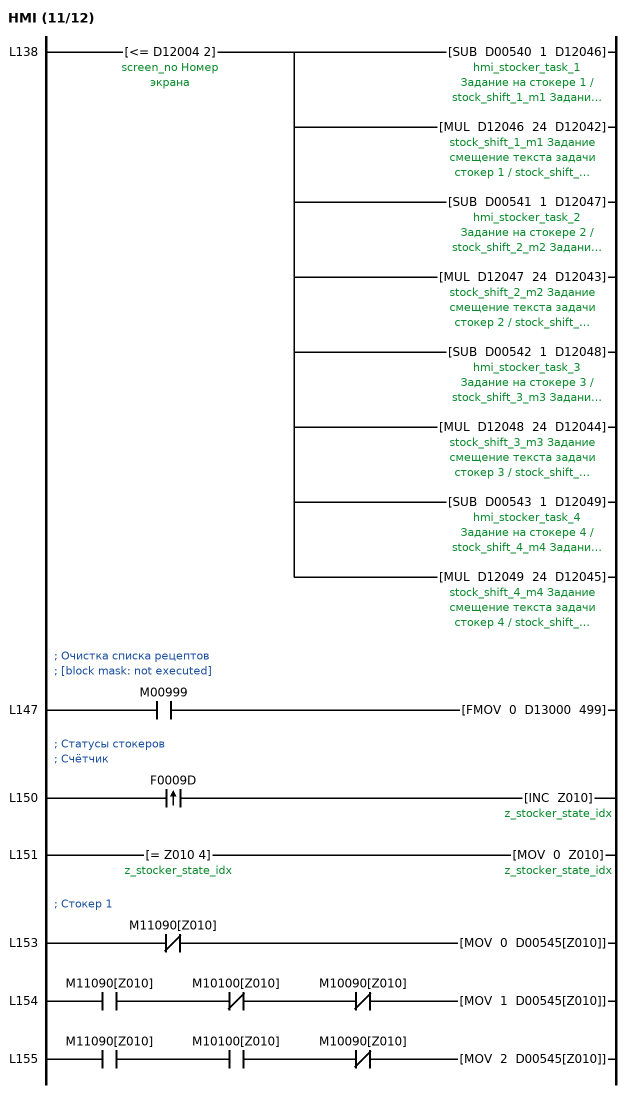
; L138
LOAD<=    D12004 2	// screen_no Номер экрана
SUB       D00540 1 D12046	// hmi_stocker_task_1 Задание на стокере 1 / stock_shift_1_m1 Задание смещение текста задачи стокер 1
MUL       D12046 24 D12042	// stock_shift_1_m1 Задание смещение текста задачи стокер 1 / stock_shift_1 Задание смещение текста задачи стокер 1
SUB       D00541 1 D12047	// hmi_stocker_task_2 Задание на стокере 2 / stock_shift_2_m2 Задание смещение текста задачи стокер 2
MUL       D12047 24 D12043	// stock_shift_2_m2 Задание смещение текста задачи стокер 2 / stock_shift_2 Задание смещение текста задачи стокер 2
SUB       D00542 1 D12048	// hmi_stocker_task_3 Задание на стокере 3 / stock_shift_3_m3 Задание смещение текста задачи стокер 3
MUL       D12048 24 D12044	// stock_shift_3_m3 Задание смещение текста задачи стокер 3 / stock_shift_3 Задание смещение текста задачи стокер 3
SUB       D00543 1 D12049	// hmi_stocker_task_4 Задание на стокере 4 / stock_shift_4_m4 Задание смещение текста задачи стокер 4
MUL       D12049 24 D12045	// stock_shift_4_m4 Задание смещение текста задачи стокер 4 / stock_shift_4 Задание смещение текста задачи стокер 4
// Очистка списка рецептов
; L147 (block mask: not executed)
LOAD      M00999
FMOV      0 D13000 499
// Статусы стокеров
// Счётчик
; L150
LOADP     F0009D
INC       Z010	// z_stocker_state_idx
; L151
LOAD=     Z010 4	// z_stocker_state_idx
MOV       0 Z010	// z_stocker_state_idx
// Стокер 1
; L153
LOAD NOT  M11090[Z010]
MOV       0 D00545[Z010]
; L154
LOAD      M11090[Z010]
AND NOT   M10100[Z010]
AND NOT   M10090[Z010]
MOV       1 D00545[Z010]
; L155
LOAD      M11090[Z010]
AND       M10100[Z010]
AND NOT   M10090[Z010]
MOV       2 D00545[Z010]

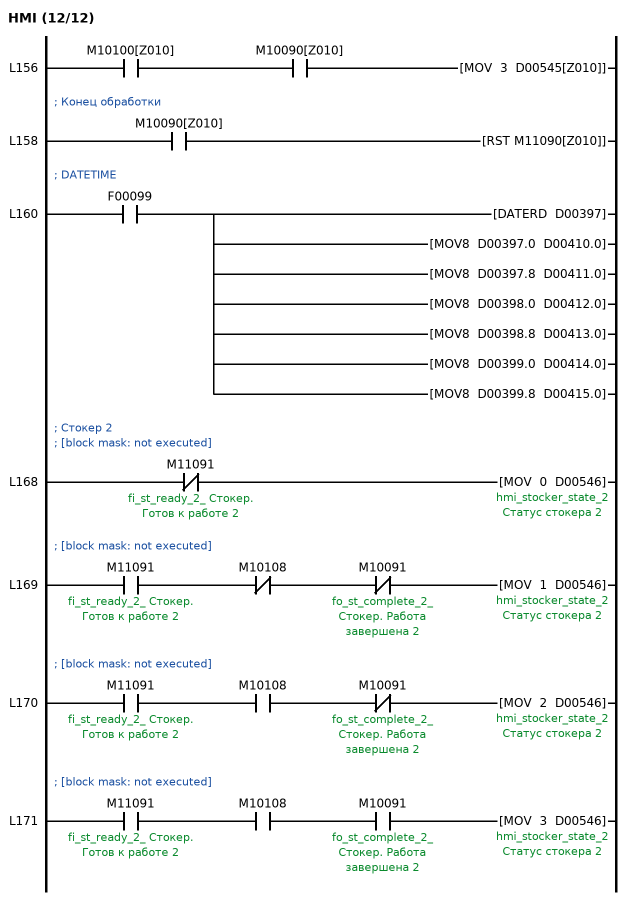
; L156
LOAD      M10100[Z010]
AND       M10090[Z010]
MOV       3 D00545[Z010]
// Конец обработки
; L158
LOAD      M10090[Z010]
RST       M11090[Z010]
// DATETIME
; L160
LOAD      F00099
DATERD    D00397
MOV8      D00397.0 D00410.0
MOV8      D00397.8 D00411.0
MOV8      D00398.0 D00412.0
MOV8      D00398.8 D00413.0
MOV8      D00399.0 D00414.0
MOV8      D00399.8 D00415.0
// Стокер 2
; L168 (block mask: not executed)
LOAD NOT  M11091	// fi_st_ready_2_ Стокер. Готов к работе 2
MOV       0 D00546	// hmi_stocker_state_2 Статус стокера 2
; L169 (block mask: not executed)
LOAD      M11091	// fi_st_ready_2_ Стокер. Готов к работе 2
AND NOT   M10108
AND NOT   M10091	// fo_st_complete_2_ Стокер. Работа завершена 2
MOV       1 D00546	// hmi_stocker_state_2 Статус стокера 2
; L170 (block mask: not executed)
LOAD      M11091	// fi_st_ready_2_ Стокер. Готов к работе 2
AND       M10108
AND NOT   M10091	// fo_st_complete_2_ Стокер. Работа завершена 2
MOV       2 D00546	// hmi_stocker_state_2 Статус стокера 2
; L171 (block mask: not executed)
LOAD      M11091	// fi_st_ready_2_ Стокер. Готов к работе 2
AND       M10108
AND       M10091	// fo_st_complete_2_ Стокер. Работа завершена 2
MOV       3 D00546	// hmi_stocker_state_2 Статус стокера 2

PROGRAM ERROR (task: Scan Program)

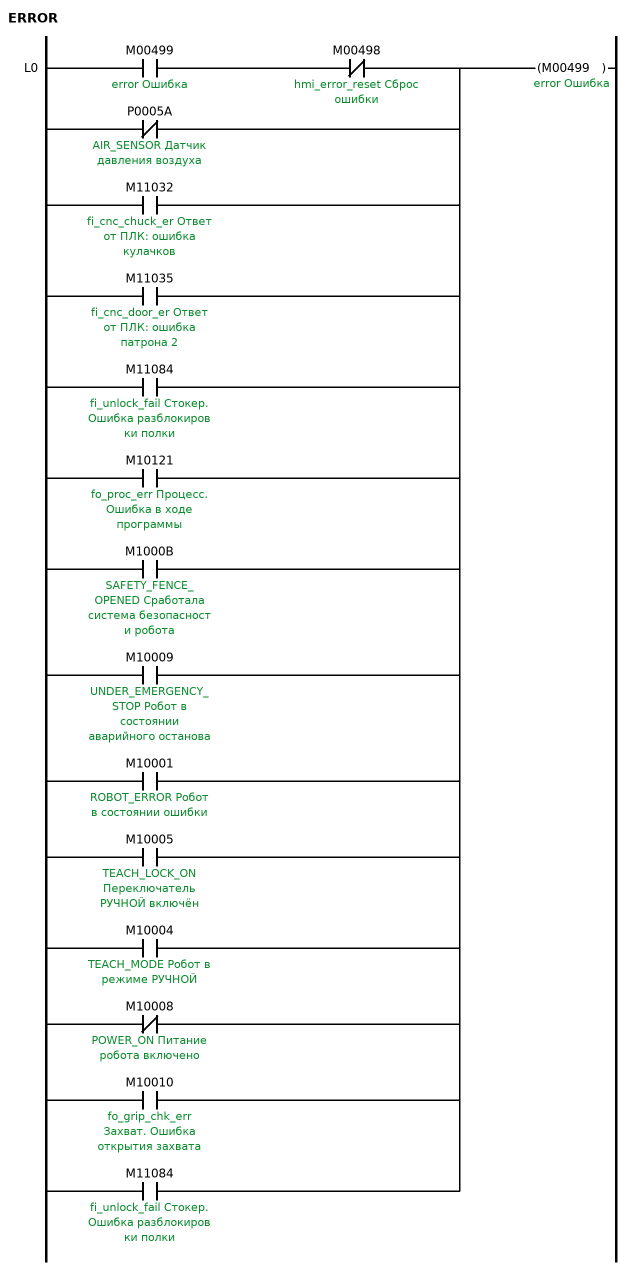
; L0
LOAD      M00499	// error Ошибка
AND NOT   M00498	// hmi_error_reset Сброс ошибки
OR NOT    P0005A	// AIR_SENSOR Датчик давления воздуха
OR        M11032	// fi_cnc_chuck_er Ответ от ПЛК: ошибка кулачков
OR        M11035	// fi_cnc_door_er Ответ от ПЛК: ошибка патрона 2
OR        M11084	// fi_unlock_fail Стокер. Ошибка разблокировки полки
OR        M10121	// fo_proc_err Процесс. Ошибка в ходе программы
OR        M1000B	// SAFETY_FENCE_OPENED Сработала система безопасности робота
OR        M10009	// UNDER_EMERGENCY_STOP Робот в состоянии аварийного останова
OR        M10001	// ROBOT_ERROR Робот в состоянии ошибки
OR        M10005	// TEACH_LOCK_ON Переключатель РУЧНОЙ включён
OR        M10004	// TEACH_MODE Робот в режиме РУЧНОЙ
OR NOT    M10008	// POWER_ON Питание робота включено
OR        M10010	// fo_grip_chk_err Захват. Ошибка открытия захвата
OR        M11084	// fi_unlock_fail Стокер. Ошибка разблокировки полки
OUT       M00499	// error Ошибка

VARIABLES AND COMMENTS (devices not used above)
M1000C	BIT	BATTERY_ALARM // Батарейка энкодеров садится
M00546	BIT	CMD_CHUCK_CLOSE // Закрыть патрон 1
P00092	BIT	CMD_LAST // Последняя деталь
P00091	BIT	CMD_RBTALM // Ошибка робота
M00513	BIT	cnc_chuck_close_flag // Флаг закрытия кулачков
M00512	BIT	cnc_chuck_open_flag // Флаг открытия кулачков
P00044	BIT	CNC_DOOR_CLOSED // Патрон 2 закрыт
P00043	BIT	CNC_DOOR_OPENED // Патрон 2 открыт
P0005F	BIT	CNC_PG_NG // Ошибка поиска программы
P00046	BIT	CNC_PG_OK // Поиск программы успешен
D00200	WORD	current_stocker
P0008F	BIT	EMPTY
M11001	BIT	EXT_ERROR_RESET // Сбросить ошибку на роботе
M11037	BIT	fi_cnc_blocked // Ответ от ПЛК: станок заблокирован
M11034	BIT	fi_cnc_door_cl // Ответ от ПЛК: патрон 2 закрыта
M11033	BIT	fi_cnc_door_op // Ответ от ПЛК: патрон 2 открыт
M1107F	BIT	fi_cnc_pick_ovp_7_ // Станок. Прижим при взятии бит 7
M11077	BIT	fi_cnc_put_ovp_7_ // Станок. Прижим при установке бит 7
M11150	BIT	fi_de_data_0_ // Обмен данными. Данные бит 0
M1115F	BIT	fi_de_data_15_ // Обмен данными. Данные бит 15
M11137	BIT	fi_de_recipe_7_ // Обмен данными. Тип рецепта бит 7
M11147	BIT	fi_de_table_el_7_ // Обмен данными. Элемент таблицы бит 7
M1113F	BIT	fi_de_table_id_7_ // Обмен данными. Номер таблицы бит 7
M11010	BIT	fi_grip_check // Захват. Проверять ли датчик открытия захвата
M11012	BIT	fi_grip_close_1_ // Захват. Закрыть захват 1
M11014	BIT	fi_grip_close_2_ // Захват. Закрыть захват 2
M1102F	BIT	fi_grip_ctime_7_ // Захват. Время на закрытие захвата бит 7
M1101C	BIT	fi_grip_etime_7_ // Захват. Время проверки захвата бит 7
M11011	BIT	fi_grip_open_1_ // Захват. Открыть захват 1
M11013	BIT	fi_grip_open_2_ // Захват. Открыть захват 2
M11027	BIT	fi_grip_otime_7_ // Захват. Время на открытие захвата бит 7
M11160	BIT	fi_mon_speed_0_ // Робот. Множитель скорости  бит 0
M11167	BIT	fi_mon_speed_7_ // Робот. Множитель скорости  бит 7
M11120	BIT	fi_proc_start // Процесс. Запуск процесса / продолжить процесс
M11127	BIT	fi_robot_pgreset // Сброс цикла
M11090	BIT	fi_st_ready_1_ // Стокер. Готов к работе 1
M11092	BIT	fi_st_ready_3_ // Стокер. Готов к работе 3
M11093	BIT	fi_st_ready_4_ // Стокер. Готов к работе 4
M1108F	BIT	fi_st_search // Стокер. Активировать подсчёт заготовок
M11107	BIT	fi_st_task_1__7_ // Процесс. Задание на стокере 1 бит 7
M1110F	BIT	fi_st_task_2__7_ // Процесс. Задание на стокере 2 бит 7
M11117	BIT	fi_st_task_3__7_ // Процесс. Задание на стокере 3 бит 7
M1111F	BIT	fi_st_task_4__7_ // Процесс. Задание на стокере 4 бит 7
M11040	BIT	fi_x_cor_cnc_0_ // Станок. Корректировка патрона по оси Х бит 0
M1104F	BIT	fi_x_cor_cnc_15_ // Станок. Корректировка патрона по оси Х бит 15
M11050	BIT	fi_y_cor_cnc_0_ // Станок. Корректировка патрона по оси Y бит 0
M1105F	BIT	fi_y_cor_cnc_15_ // Станок. Корректировка патрона по оси Y бит 15
M11060	BIT	fi_z_cor_cnc_0_ // Станок. Корректировка патрона по оси Z бит 0
M1106F	BIT	fi_z_cor_cnc_15_ // Станок. Корректировка патрона по оси Z бит 15
M12022	BIT	flag_load_type_6 // Флаг загруить элемент типа 6
M12023	BIT	flag_load_type_7 // Флаг загруить элемент типа 7
M12024	BIT	flag_load_type_8 // Флаг загруить элемент типа 8
M1201A	BIT	flag_save_type_6 // Флаг сохранить элемент типа 6
M1201B	BIT	flag_save_type_7 // Флаг сохранить элемент типа 7
M1201C	BIT	flag_save_type_8 // Флаг сохранить элемент типа 8
M10037	BIT	fo_cnc_block // Команда станку - заблокировать
M1003F	BIT	fo_cnc_pg_7_ // Команда станку - бит программы 7
M10012	BIT	fo_grip_closed_1_ // Захват. Захват 1 закрыт
M10014	BIT	fo_grip_closed_2_ // Захват. Захват 2 закрыт
M10011	BIT	fo_grip_opened_1_ // Захват. Захват 1 открыт
M10013	BIT	fo_grip_opened_2_ // Захват. Захват 2 открыт
M10015	BIT	fo_grip_sensor // Захват. Датчик заготовки
M10120	BIT	fo_proc_on // Процесс. Процесс запущен
M10090	BIT	fo_st_complete_1_ // Стокер. Работа завершена 1
M10092	BIT	fo_st_complete_3_ // Стокер. Работа завершена 3
M10093	BIT	fo_st_complete_4_ // Стокер. Работа завершена 4
M10085	BIT	fo_st_opened_1_ // Стокер. Открыт 1
M10086	BIT	fo_st_opened_2_ // Стокер. Открыт 2
M10087	BIT	fo_st_opened_3_ // Стокер. Открыт 3
M10088	BIT	fo_st_opened_4_ // Стокер. Открыт 4
M00551	BIT	hmi_air_off
D00512	WORD	hmi_chuck_close_time // Время на закрытие кулачков
D00513	WORD	hmi_chuck_err_time // Время ошибки кулачков
D00511	WORD	hmi_chuck_open_time // Время на открытие кулачков
M0050A	BIT	hmi_cnc_chuck_close_check // Проверять датчик закрытия кулачков станка
M00509	BIT	hmi_cnc_chuck_open_check // Проверять датчик открытия кулачков станка
M0050E	BIT	hmi_cnc_door_close_check // Проверять датчик закрытия патрона 2 станка
M0050D	BIT	hmi_cnc_door_open_check // Проверять датчик открытия патрона 2 станка
M00516	BIT	hmi_cnc_lock // Команда станку с HMI  - заблокировать
D00522	WORD	hmi_cnc_pick_ovlp // Оверлап при взятии 
D00523	WORD	hmi_cnc_put_ovlp // Оверлап при заборе
M00517	BIT	hmi_cnc_unlock // Команда станку с HMI  - разблокировать
D00519	WORD	hmi_cnc_x_cor // Корректировка точки станка Х
D00520	WORD	hmi_cnc_y_cor // Корректировка точки станка Y
D00521	WORD	hmi_cnc_z_cor // Корректировка точки станка Z
M0052B	BIT	hmi_door_chuck_close // Лампа Датчик закрытия патрона 2
M0052A	BIT	hmi_door_chuck_open // Лампа Датчик открытия патрона 2
D00516	WORD	hmi_door_close_time // Время на закрытие патрона 2
D00517	WORD	hmi_door_err_time // Время ошибки патрона 2
D00515	WORD	hmi_door_open_time // Время на открытие патрона 2
M00529	BIT	hmi_lamp_chuck_close // Лампа Датчик закрытия кулачков
M00528	BIT	hmi_lamp_chuck_open // Лампа Датчик открытия кулачков
M00525	BIT	hmi_robot_process_on // Запуск процесса обработки 
M00526	BIT	hmi_robot_process_stop // Остановка процесса обработки 
M00506	BIT	hmi_robot_slow // Замедление робота при приближении
D12624.0	BIT	hmi_shaft_back // Требуется ли возврат вала в кондуктор
D00534	WORD	hmi_stocker_open_delay // Задержка при открытии стокера
D00545	WORD	hmi_stocker_state_1 // Статус стокера 1
D00547	WORD	hmi_stocker_state_3 // Статус стокера 3
D00548	WORD	hmi_stocker_state_4 // Статус стокера 4
M10006	BIT	HOME // Робот в домашнем положении 1
M10007	BIT	HOME2 // Робот в домашнем положении 2
D12050	WORD	plate_name_shift // Смещение имени пластины коррекция
D12051	WORD	plate_name_shift_m1 // Смещение имени пластины коррекция
D00500	WORD	plc_power_errors // Количество включений ПЛК 
D12001	WORD	recipe_error_code // Код ошибки рецепта
M12002	BIT	recipe_state_ok // Рецепт сохранён/загружен
M12012	BIT	save_ok_type_6 // Элемент сохранён тип 6
M12013	BIT	save_ok_type_7 // Элемент сохранён тип 7
M12014	BIT	save_ok_type_8 // Элемент сохранён тип 8
M1200A	BIT	save_type_6 // Сохранить элемент типа 6
M1200B	BIT	save_type_7 // Сохранить элемент типа 7
M1200C	BIT	save_type_8 // Сохранить элемент типа 8
M00000	BIT	start_task
T0560	BIT/WORD	T100_data_ready_1 // Таймер на подготовку данных 1
T0561	BIT/WORD	T100_data_ready_2 // Таймер на подготовку данных 2
T0562	BIT/WORD	T100_data_ready_3 // Таймер на подготовку данных 3
T0563	BIT/WORD	T100_data_ready_4 // Таймер на подготовку данных 4
T0564	BIT/WORD	T100_data_ready_5 // Таймер на подготовку данных 5
T0565	BIT/WORD	T100_data_ready_6 // Таймер на подготовку данных 6
T0566	BIT/WORD	T100_data_ready_7 // Таймер на подготовку данных 7
T0921	BIT/WORD	T100_load_delay_6 // Таймаут на загрузку 6
T0922	BIT/WORD	T100_load_delay_7 // Таймаут на загрузку 7
T0913	BIT/WORD	T100_save_delay_6 // Время сохранения 6
T0914	BIT/WORD	T100_save_delay_7 // Время сохранения 7
T0915	BIT/WORD	T100_save_delay_8 // Время сохранения 8
M00001	BIT	work_stocker_1
M00002	BIT	work_stocker_2
M00003	BIT	work_stocker_3
M00004	BIT	work_stocker_4
M10039	BIT	Команда станку - бит программы 1
M1003A	BIT	Команда станку - бит программы 2
M1003B	BIT	Команда станку - бит программы 3
M1003C	BIT	Команда станку - бит программы 4
M1003D	BIT	Команда станку - бит программы 5
M1003E	BIT	Команда станку - бит программы 6
M11016	BIT	Захват. Время проверки захвата бит 1
M11017	BIT	Захват. Время проверки захвата бит 2
M11018	BIT	Захват. Время проверки захвата бит 3
M11019	BIT	Захват. Время проверки захвата бит 4
M1101A	BIT	Захват. Время проверки захвата бит 5
M1101B	BIT	Захват. Время проверки захвата бит 6
M11021	BIT	Захват. Время на открытие захвата бит 1
M11022	BIT	Захват. Время на открытие захвата бит 2
M11023	BIT	Захват. Время на открытие захвата бит 3
M11024	BIT	Захват. Время на открытие захвата бит 4
M11025	BIT	Захват. Время на открытие захвата бит 5
M11026	BIT	Захват. Время на открытие захвата бит 6
M11029	BIT	Захват. Время на закрытие захвата бит 1
M1102A	BIT	Захват. Время на закрытие захвата бит 2
M1102B	BIT	Захват. Время на закрытие захвата бит 3
M1102C	BIT	Захват. Время на закрытие захвата бит 4
M1102D	BIT	Захват. Время на закрытие захвата бит 5
M1102E	BIT	Захват. Время на закрытие захвата бит 6
M11041	BIT	Станок. Корректировка патрона по оси Х бит 1
M11042	BIT	Станок. Корректировка патрона по оси Х бит 2
M11043	BIT	Станок. Корректировка патрона по оси Х бит 3
M11044	BIT	Станок. Корректировка патрона по оси Х бит 4
M11045	BIT	Станок. Корректировка патрона по оси Х бит 5
M11046	BIT	Станок. Корректировка патрона по оси Х бит 6
M11047	BIT	Станок. Корректировка патрона по оси Х бит 7
M11048	BIT	Станок. Корректировка патрона по оси Х бит 8
M11049	BIT	Станок. Корректировка патрона по оси Х бит 9
M1104A	BIT	Станок. Корректировка патрона по оси Х бит 10
M1104B	BIT	Станок. Корректировка патрона по оси Х бит 11
M1104C	BIT	Станок. Корректировка патрона по оси Х бит 12
M1104D	BIT	Станок. Корректировка патрона по оси Х бит 13
M1104E	BIT	Станок. Корректировка патрона по оси Х бит 14
M11051	BIT	Станок. Корректировка патрона по оси Y бит 1
M11052	BIT	Станок. Корректировка патрона по оси Y бит 2
M11053	BIT	Станок. Корректировка патрона по оси Y бит 3
M11054	BIT	Станок. Корректировка патрона по оси Y бит 4
M11055	BIT	Станок. Корректировка патрона по оси Y бит 5
M11056	BIT	Станок. Корректировка патрона по оси Y бит 6
M11057	BIT	Станок. Корректировка патрона по оси Y бит 7
M11058	BIT	Станок. Корректировка патрона по оси Y бит 8
M11059	BIT	Станок. Корректировка патрона по оси Y бит 9
M1105A	BIT	Станок. Корректировка патрона по оси Y бит 10
M1105B	BIT	Станок. Корректировка патрона по оси Y бит 11
M1105C	BIT	Станок. Корректировка патрона по оси Y бит 12
M1105D	BIT	Станок. Корректировка патрона по оси Y бит 13
M1105E	BIT	Станок. Корректировка патрона по оси Y бит 14
M11061	BIT	Станок. Корректировка патрона по оси Z бит 1
M11062	BIT	Станок. Корректировка патрона по оси Z бит 2
M11063	BIT	Станок. Корректировка патрона по оси Z бит 3
M11064	BIT	Станок. Корректировка патрона по оси Z бит 4
M11065	BIT	Станок. Корректировка патрона по оси Z бит 5
M11066	BIT	Станок. Корректировка патрона по оси Z бит 6
M11067	BIT	Станок. Корректировка патрона по оси Z бит 7
M11068	BIT	Станок. Корректировка патрона по оси Z бит 8
M11069	BIT	Станок. Корректировка патрона по оси Z бит 9
M1106A	BIT	Станок. Корректировка патрона по оси Z бит 10
M1106B	BIT	Станок. Корректировка патрона по оси Z бит 11
M1106C	BIT	Станок. Корректировка патрона по оси Z бит 12
M1106D	BIT	Станок. Корректировка патрона по оси Z бит 13
M1106E	BIT	Станок. Корректировка патрона по оси Z бит 14
M11071	BIT	Станок. Прижим при установке бит 1
M11072	BIT	Станок. Прижим при установке бит 2
M11073	BIT	Станок. Прижим при установке бит 3
M11074	BIT	Станок. Прижим при установке бит 4
M11075	BIT	Станок. Прижим при установке бит 5
M11076	BIT	Станок. Прижим при установке бит 6
M11079	BIT	Станок. Прижим при взятии бит 1
M1107A	BIT	Станок. Прижим при взятии бит 2
M1107B	BIT	Станок. Прижим при взятии бит 3
M1107C	BIT	Станок. Прижим при взятии бит 4
M1107D	BIT	Станок. Прижим при взятии бит 5
M1107E	BIT	Станок. Прижим при взятии бит 6
M11101	BIT	Процесс. Задание на стокере 1 бит 1
M11102	BIT	Процесс. Задание на стокере 1 бит 2
M11103	BIT	Процесс. Задание на стокере 1 бит 3
M11104	BIT	Процесс. Задание на стокере 1 бит 4
M11105	BIT	Процесс. Задание на стокере 1 бит 5
M11106	BIT	Процесс. Задание на стокере 1 бит 6
M11109	BIT	Процесс. Задание на стокере 2 бит 1
M1110A	BIT	Процесс. Задание на стокере 2 бит 2
M1110B	BIT	Процесс. Задание на стокере 2 бит 3
M1110C	BIT	Процесс. Задание на стокере 2 бит 4
M1110D	BIT	Процесс. Задание на стокере 2 бит 5
M1110E	BIT	Процесс. Задание на стокере 2 бит 6
M11111	BIT	Процесс. Задание на стокере 3 бит 1
M11112	BIT	Процесс. Задание на стокере 3 бит 2
M11113	BIT	Процесс. Задание на стокере 3 бит 3
M11114	BIT	Процесс. Задание на стокере 3 бит 4
M11115	BIT	Процесс. Задание на стокере 3 бит 5
M11116	BIT	Процесс. Задание на стокере 3 бит 6
M11119	BIT	Процесс. Задание на стокере 4 бит 1
M1111A	BIT	Процесс. Задание на стокере 4 бит 2
M1111B	BIT	Процесс. Задание на стокере 4 бит 3
M1111C	BIT	Процесс. Задание на стокере 4 бит 4
M1111D	BIT	Процесс. Задание на стокере 4 бит 5
M1111E	BIT	Процесс. Задание на стокере 4 бит 6
M11131	BIT	Обмен данными. Тип рецепта бит 1
M11132	BIT	Обмен данными. Тип рецепта бит 2
M11133	BIT	Обмен данными. Тип рецепта бит 3
M11134	BIT	Обмен данными. Тип рецепта бит 4
M11135	BIT	Обмен данными. Тип рецепта бит 5
M11136	BIT	Обмен данными. Тип рецепта бит 6
M11139	BIT	Обмен данными. Номер таблицы бит 1
M1113A	BIT	Обмен данными. Номер таблицы бит 2
M1113B	BIT	Обмен данными. Номер таблицы бит 3
M1113C	BIT	Обмен данными. Номер таблицы бит 4
M1113D	BIT	Обмен данными. Номер таблицы бит 5
M1113E	BIT	Обмен данными. Номер таблицы бит 6
M11141	BIT	Обмен данными. Элемент таблицы бит 1
M11142	BIT	Обмен данными. Элемент таблицы бит 2
M11143	BIT	Обмен данными. Элемент таблицы бит 3
M11144	BIT	Обмен данными. Элемент таблицы бит 4
M11145	BIT	Обмен данными. Элемент таблицы бит 5
M11146	BIT	Обмен данными. Элемент таблицы бит 6
M11151	BIT	Обмен данными. Данные бит 1
M11152	BIT	Обмен данными. Данные бит 2
M11153	BIT	Обмен данными. Данные бит 3
M11154	BIT	Обмен данными. Данные бит 4
M11155	BIT	Обмен данными. Данные бит 5
M11156	BIT	Обмен данными. Данные бит 6
M11157	BIT	Обмен данными. Данные бит 7
M11158	BIT	Обмен данными. Данные бит 8
M11159	BIT	Обмен данными. Данные бит 9
M1115A	BIT	Обмен данными. Данные бит 10
M1115B	BIT	Обмен данными. Данные бит 11
M1115C	BIT	Обмен данными. Данные бит 12
M1115D	BIT	Обмен данными. Данные бит 13
M1115E	BIT	Обмен данными. Данные бит 14
M11161	BIT	Робот. Множитель скорости  бит 1
M11162	BIT	Робот. Множитель скорости  бит 2
M11163	BIT	Робот. Множитель скорости  бит 3
M11164	BIT	Робот. Множитель скорости  бит 4
M11165	BIT	Робот. Множитель скорости  бит 5
M11166	BIT	Робот. Множитель скорости  бит 6